TYPE ST_System_HOHW_Stellwert :
STRUCT
	Anford_Stellventil		: BOOL;
	Anford_Pumpe		: BOOL;
	Freigabe_Anlage		: BOOL;
END_STRUCT
END_TYPE

(* stored: Version 1.1.0.1, ProductVersion 3.1.4024.9
   DUT ST_System_HOHW_Stellwert: Id {f43d615e-321e-4bac-949b-3f9c5e3175d6} *)
